// TIA Portal V17 export
// export: Created 2026-04-13T11:12:44.9491933Z, ExportSetting WithDefaults, DisplayName Totally Integrated Automation Portal, DisplayVersion V17 Update 4, DisplayName TIA Portal Openness, DisplayVersion V17 Update 4, DisplayName TIA Portal Version Control Interface, DisplayVersion V17, DisplayName SINAMICS Startdrive Advanced, DisplayVersion V17, DisplayName SINAMICS Startdrive G130, G150, S120, S150, SINAMICS MV, S210, DisplayVersion V17, DisplayName SINAMICS Startdrive G110M, G120, G120C, G120D, G120P, G115D, DisplayVersion V17, DisplayName STEP 7 Professional, DisplayVersion V17 Update 4, DisplayName STEP 7 Safety, DisplayVersion V17, DisplayName WinCC Professional, DisplayVersion V17 Update 4
FUNCTION_BLOCK "Receive_P2P"   // FB614, SCL
TITLE = Receive Data
AUTHOR : SIMATIC
FAMILY : Freeport
NAME : RcvP2P
VERSION : 4.1
// stored: IsIECCheckEnabled true, SetENOAutomatically false, UDAEnableTagReadback false
   VAR_INPUT
      PORT : PORT := 16#0000;   // Kommunikationsport, Hardwarekennung / Communication port, Hardware Identifier
      BUFFER : Variant;   // Referenz auf den Empfangspuffer / Reference to the receive buffer
   END_VAR
   VAR_OUTPUT
      UNIVERSAL : Bool;   // Access mode of communication module. 0 = universal, 1 = performance
      NDR : Bool;   // Neue Daten empfangen / New data received
      LENGTH : UInt := 16#0000;   // Länge der empfangenen Daten in Byte / Length of the current received message in bytes
      ERROR : Bool;   // Anweisung beendet mit Fehler / Instruction finished with error
      STATUS : Word := W#16#7000;   // Zusätzliche Fehlerinformation / Detailed error information
   END_VAR
   VAR
      OldPORT : PORT;   // Gespeicherter Wert für den Kommunikationsport, / Save value for Communication port
      received_length : UInt := 0;   // empfangene Länge / Received length
      y_ptp_status : SInt;   // Nur für internen Gebrauch / For internal use only
      y_state : SInt := 0;   // Status der Anweisung / State of instruction
      y_seq_nr : Byte := B#16#00;   // Sequenznummer der empfangenen Datensätze / Sequence number of data records
      safe_h1 : Byte;   // Nur für internen Gebrauch / For internal use only
      safe_h2 : Byte;   // Nur für internen Gebrauch / For internal use only
      safe_h3 : Byte;   // Nur für internen Gebrauch / For internal use only
      safe_h4 : Byte;   // Nur für internen Gebrauch / For internal use only
      isClassic : Bool;   // Nur für internen Gebrauch / For internal use only
      record_nr : Int := 49;   // Nur für internen Gebrauch / For internal use only
      offset : UDInt;   // Nur für internen Gebrauch / For internal use only
      RDREC { S7_SetPoint := 'True'} : RDREC;   // Lokale Instanz der Anweisung RDREC / Local instance of instruction RDREC
   END_VAR
   VAR DB_SPECIFIC
      ReceiveBuffer : Array[0..1027] of Byte;   // Nur für internen Gebrauch / For internal use only
   END_VAR
   VAR
      i_addr : UDInt;   // IO Adresse des Moduls / IO address of the module
      o_addr { ExternalAccessible := 'False'; ExternalVisible := 'False'; ExternalWritable := 'False'} : UDInt;
   END_VAR
BEGIN
END_FUNCTION_BLOCK
